PROGRAM prg_ProductenTellen
VAR
	bSensor		AT		%I*		:BOOL;
	
	bKlep		AT		%Q*		:BOOL; //0 is rechtdoor, 1 is afgebogen
	CounterRechtdoor: CTU;
	CounterAfslaan: CTU;
END_VAR

IF 	NOT(bKlep) THEN
CounterRechtdoor(
	CU:= bSensor, 
	PV:= 10);
END_IF

IF CounterRechtdoor.Q THEN
	bKlep := 1;
	CounterRechtdoor.RESET := TRUE;
END_IF

IF bKlep THEN
CounterAfslaan(
	CU:= bSensor,  
	PV:= 20,);
END_IF

IF CounterAfslaan.Q THEN
	bKlep := 0;
	CounterAfslaan.RESET := TRUE;
END_IF

END_PROGRAM

(* stored: Version 1.1.0.1, ProductVersion 3.1.4024.15
   POU prg_ProductenTellen: Id {e18161f0-894e-406c-a80f-4b6353825cb2}, SpecialFunc None *)
